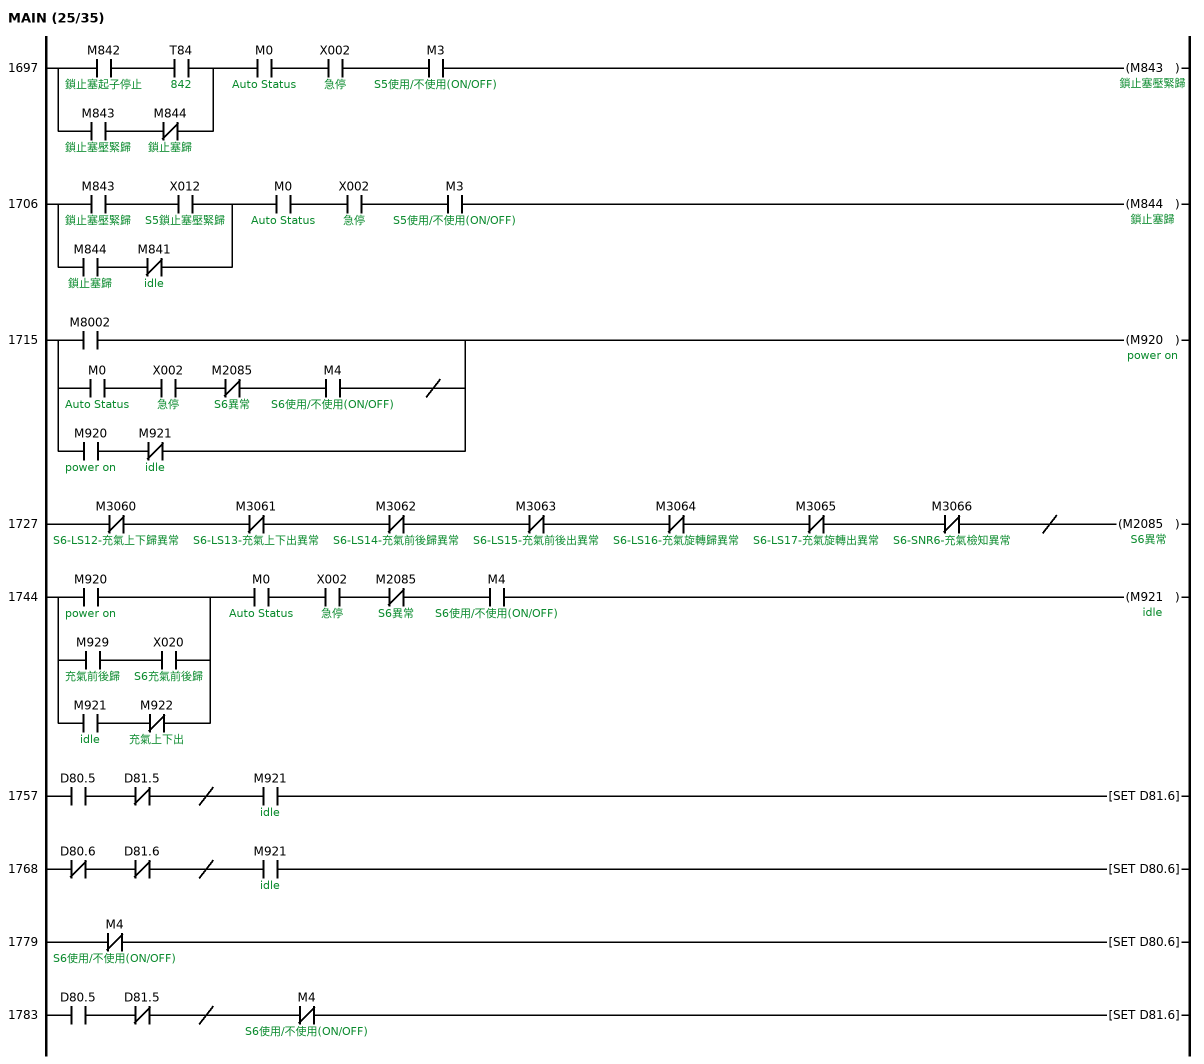
[picture p24: ladder of MAIN, rungs at steps 1697 to 1783]
1697  LD      M842  ; 鎖止塞起子停止
      AND     T84  ; 842
      LD      M843  ; 鎖止塞壓緊歸
      ANI     M844  ; 鎖止塞歸
      ORB
      AND     M0  ; Auto Status
      AND     X002  ; 急停
      AND     M3  ; S5使用/不使用(ON/OFF)
      OUT     M843  ; 鎖止塞壓緊歸
1706  LD      M843  ; 鎖止塞壓緊歸
      AND     X012  ; S5鎖止塞壓緊歸
      LD      M844  ; 鎖止塞歸
      ANI     M841  ; idle
      ORB
      AND     M0  ; Auto Status
      AND     X002  ; 急停
      AND     M3  ; S5使用/不使用(ON/OFF)
      OUT     M844  ; 鎖止塞歸
1715  LD      M8002
      LD      M0  ; Auto Status
      AND     X002  ; 急停
      ANI     M2085  ; S6異常
      AND     M4  ; S6使用/不使用(ON/OFF)
      INV
      ORB
      LD      M920  ; power on
      ANI     M921  ; idle
      ORB
      OUT     M920  ; power on
1727  LDI     M3060  ; S6-LS12-充氣上下歸異常
      ANI     M3061  ; S6-LS13-充氣上下出異常
      ANI     M3062  ; S6-LS14-充氣前後歸異常
      ANI     M3063  ; S6-LS15-充氣前後出異常
      ANI     M3064  ; S6-LS16-充氣旋轉歸異常
      ANI     M3065  ; S6-LS17-充氣旋轉出異常
      ANI     M3066  ; S6-SNR6-充氣檢知異常
      INV
      OUT     M2085  ; S6異常
1744  LD      M920  ; power on
      LD      M929  ; 充氣前後歸
      AND     X020  ; S6充氣前後歸
      ORB
      LD      M921  ; idle
      ANI     M922  ; 充氣上下出
      ORB
      AND     M0  ; Auto Status
      AND     X002  ; 急停
      ANI     M2085  ; S6異常
      AND     M4  ; S6使用/不使用(ON/OFF)
      OUT     M921  ; idle
1757  LD      D80.5
      ANI     D81.5
      INV
      AND     M921  ; idle
      SET     D81.6
1768  LDI     D80.6
      ANI     D81.6
      INV
      AND     M921  ; idle
      SET     D80.6
1779  LDI     M4  ; S6使用/不使用(ON/OFF)
      SET     D80.6
1783  LD      D80.5
      ANI     D81.5
      INV
      ANI     M4  ; S6使用/不使用(ON/OFF)
      SET     D81.6
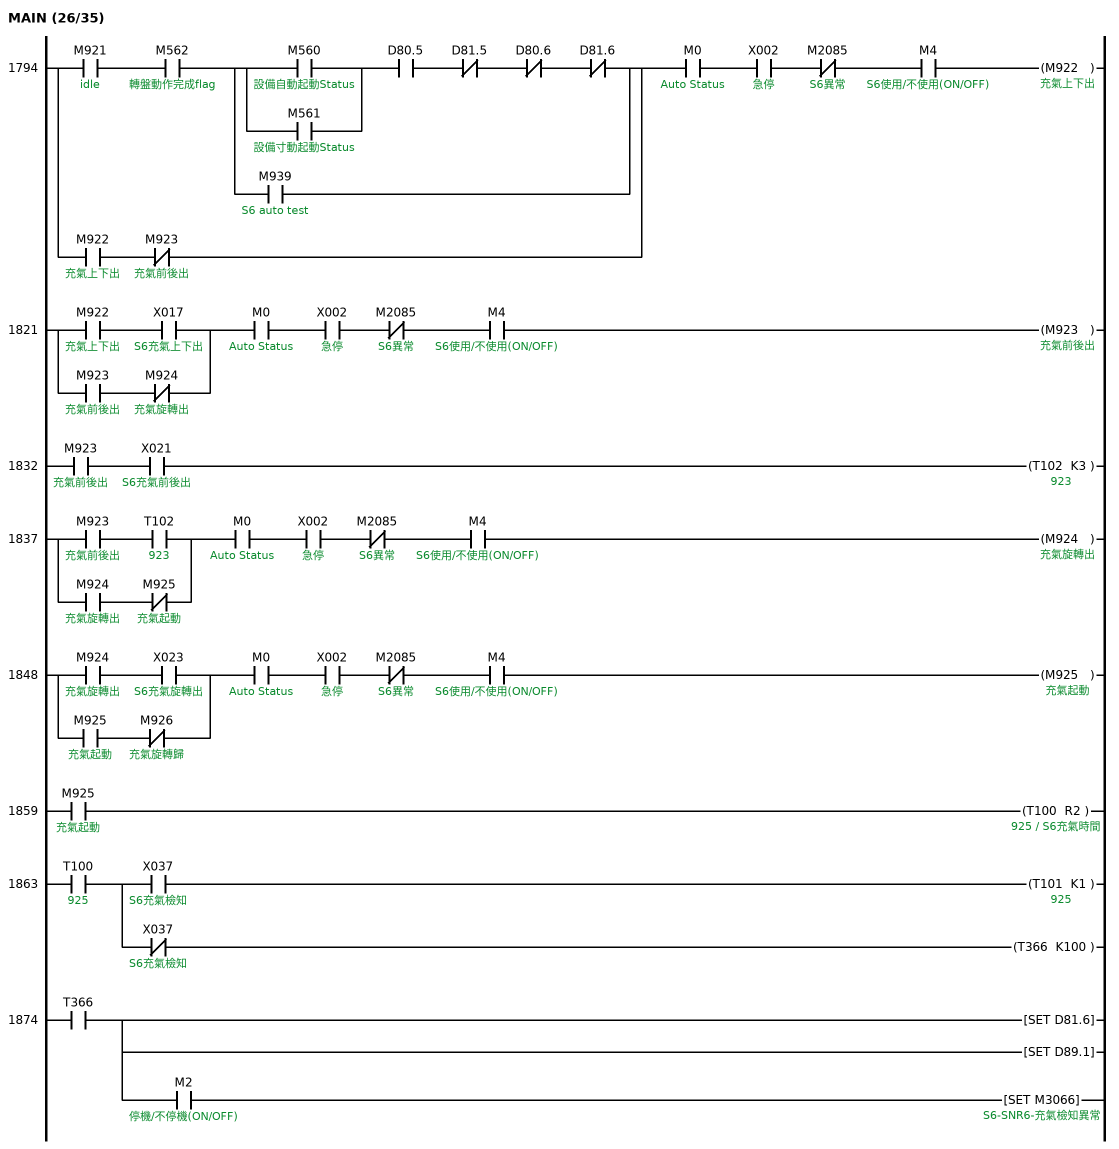
1794  LD      M921  ; idle
      AND     M562  ; 轉盤動作完成flag
      LD      M560  ; 設備自動起動Status
      OR      M561  ; 設備寸動起動Status
      AND     D80.5
      ANI     D81.5
      ANI     D80.6
      ANI     D81.6
      OR      M939  ; S6 auto test
      ANB
      LD      M922  ; 充氣上下出
      ANI     M923  ; 充氣前後出
      ORB
      AND     M0  ; Auto Status
      AND     X002  ; 急停
      ANI     M2085  ; S6異常
      AND     M4  ; S6使用/不使用(ON/OFF)
      OUT     M922  ; 充氣上下出
1821  LD      M922  ; 充氣上下出
      AND     X017  ; S6充氣上下出
      LD      M923  ; 充氣前後出
      ANI     M924  ; 充氣旋轉出
      ORB
      AND     M0  ; Auto Status
      AND     X002  ; 急停
      ANI     M2085  ; S6異常
      AND     M4  ; S6使用/不使用(ON/OFF)
      OUT     M923  ; 充氣前後出
1832  LD      M923  ; 充氣前後出
      AND     X021  ; S6充氣前後出
      OUT     T102 K3  ; 923
1837  LD      M923  ; 充氣前後出
      AND     T102  ; 923
      LD      M924  ; 充氣旋轉出
      ANI     M925  ; 充氣起動
      ORB
      AND     M0  ; Auto Status
      AND     X002  ; 急停
      ANI     M2085  ; S6異常
      AND     M4  ; S6使用/不使用(ON/OFF)
      OUT     M924  ; 充氣旋轉出
1848  LD      M924  ; 充氣旋轉出
      AND     X023  ; S6充氣旋轉出
      LD      M925  ; 充氣起動
      ANI     M926  ; 充氣旋轉歸
      ORB
      AND     M0  ; Auto Status
      AND     X002  ; 急停
      ANI     M2085  ; S6異常
      AND     M4  ; S6使用/不使用(ON/OFF)
      OUT     M925  ; 充氣起動
1859  LD      M925  ; 充氣起動
      OUT     T100 R2  ; 925 / S6充氣時間
1863  LD      T100  ; 925
      MPS
      AND     X037  ; S6充氣檢知
      OUT     T101 K1  ; 925
      MPP
      ANI     X037  ; S6充氣檢知
      OUT     T366 K100
1874  LD      T366
      SET     D81.6
      SET     D89.1
      AND     M2  ; 停機/不停機(ON/OFF)
      SET     M3066  ; S6-SNR6-充氣檢知異常
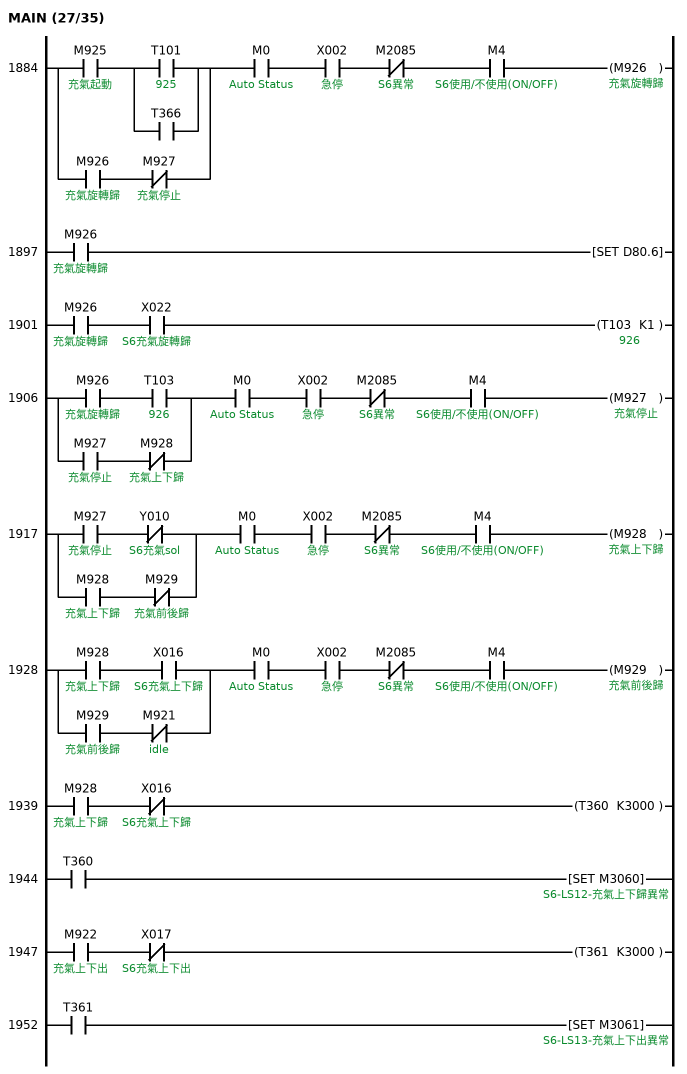
1884  LD      M925  ; 充氣起動
      LD      T101  ; 925
      OR      T366
      ANB
      LD      M926  ; 充氣旋轉歸
      ANI     M927  ; 充氣停止
      ORB
      AND     M0  ; Auto Status
      AND     X002  ; 急停
      ANI     M2085  ; S6異常
      AND     M4  ; S6使用/不使用(ON/OFF)
      OUT     M926  ; 充氣旋轉歸
1897  LD      M926  ; 充氣旋轉歸
      SET     D80.6
1901  LD      M926  ; 充氣旋轉歸
      AND     X022  ; S6充氣旋轉歸
      OUT     T103 K1  ; 926
1906  LD      M926  ; 充氣旋轉歸
      AND     T103  ; 926
      LD      M927  ; 充氣停止
      ANI     M928  ; 充氣上下歸
      ORB
      AND     M0  ; Auto Status
      AND     X002  ; 急停
      ANI     M2085  ; S6異常
      AND     M4  ; S6使用/不使用(ON/OFF)
      OUT     M927  ; 充氣停止
1917  LD      M927  ; 充氣停止
      ANI     Y010  ; S6充氣sol
      LD      M928  ; 充氣上下歸
      ANI     M929  ; 充氣前後歸
      ORB
      AND     M0  ; Auto Status
      AND     X002  ; 急停
      ANI     M2085  ; S6異常
      AND     M4  ; S6使用/不使用(ON/OFF)
      OUT     M928  ; 充氣上下歸
1928  LD      M928  ; 充氣上下歸
      AND     X016  ; S6充氣上下歸
      LD      M929  ; 充氣前後歸
      ANI     M921  ; idle
      ORB
      AND     M0  ; Auto Status
      AND     X002  ; 急停
      ANI     M2085  ; S6異常
      AND     M4  ; S6使用/不使用(ON/OFF)
      OUT     M929  ; 充氣前後歸
1939  LD      M928  ; 充氣上下歸
      ANI     X016  ; S6充氣上下歸
      OUT     T360 K3000
1944  LD      T360
      SET     M3060  ; S6-LS12-充氣上下歸異常
1947  LD      M922  ; 充氣上下出
      ANI     X017  ; S6充氣上下出
      OUT     T361 K3000
1952  LD      T361
      SET     M3061  ; S6-LS13-充氣上下出異常
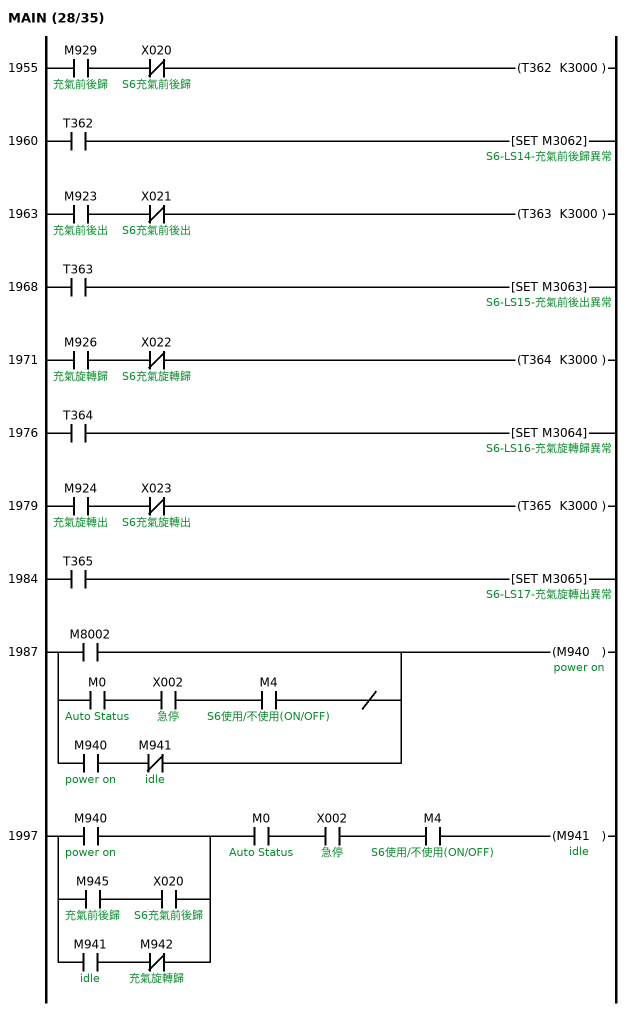
1955  LD      M929  ; 充氣前後歸
      ANI     X020  ; S6充氣前後歸
      OUT     T362 K3000
1960  LD      T362
      SET     M3062  ; S6-LS14-充氣前後歸異常
1963  LD      M923  ; 充氣前後出
      ANI     X021  ; S6充氣前後出
      OUT     T363 K3000
1968  LD      T363
      SET     M3063  ; S6-LS15-充氣前後出異常
1971  LD      M926  ; 充氣旋轉歸
      ANI     X022  ; S6充氣旋轉歸
      OUT     T364 K3000
1976  LD      T364
      SET     M3064  ; S6-LS16-充氣旋轉歸異常
1979  LD      M924  ; 充氣旋轉出
      ANI     X023  ; S6充氣旋轉出
      OUT     T365 K3000
1984  LD      T365
      SET     M3065  ; S6-LS17-充氣旋轉出異常
1987  LD      M8002
      LD      M0  ; Auto Status
      AND     X002  ; 急停
      AND     M4  ; S6使用/不使用(ON/OFF)
      INV
      ORB
      LD      M940  ; power on
      ANI     M941  ; idle
      ORB
      OUT     M940  ; power on
1997  LD      M940  ; power on
      LD      M945  ; 充氣前後歸
      AND     X020  ; S6充氣前後歸
      ORB
      LD      M941  ; idle
      ANI     M942  ; 充氣旋轉歸
      ORB
      AND     M0  ; Auto Status
      AND     X002  ; 急停
      AND     M4  ; S6使用/不使用(ON/OFF)
      OUT     M941  ; idle
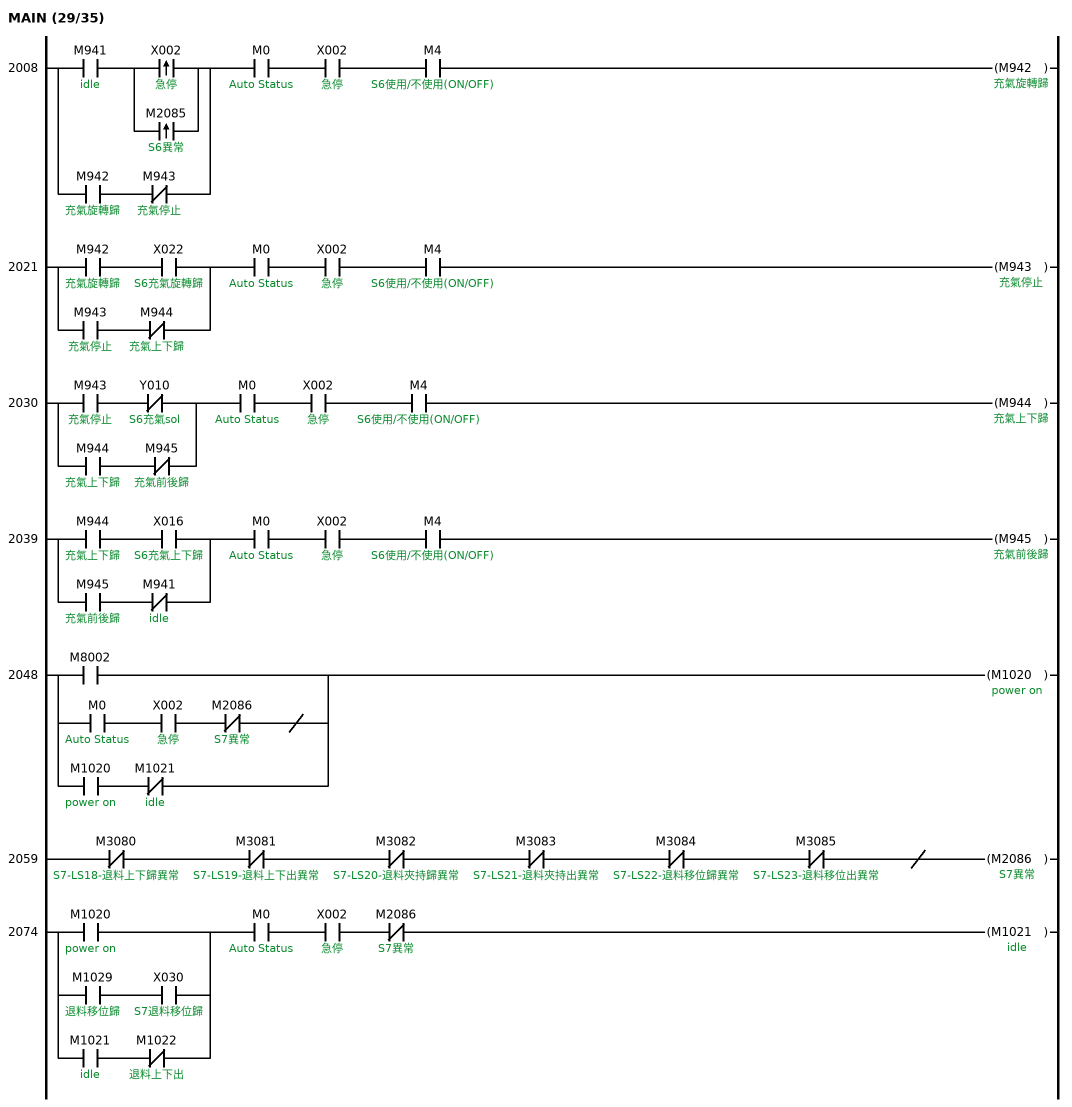
2008  LD      M941  ; idle
      LDP     X002  ; 急停
      ORP     M2085  ; S6異常
      ANB
      LD      M942  ; 充氣旋轉歸
      ANI     M943  ; 充氣停止
      ORB
      AND     M0  ; Auto Status
      AND     X002  ; 急停
      AND     M4  ; S6使用/不使用(ON/OFF)
      OUT     M942  ; 充氣旋轉歸
2021  LD      M942  ; 充氣旋轉歸
      AND     X022  ; S6充氣旋轉歸
      LD      M943  ; 充氣停止
      ANI     M944  ; 充氣上下歸
      ORB
      AND     M0  ; Auto Status
      AND     X002  ; 急停
      AND     M4  ; S6使用/不使用(ON/OFF)
      OUT     M943  ; 充氣停止
2030  LD      M943  ; 充氣停止
      ANI     Y010  ; S6充氣sol
      LD      M944  ; 充氣上下歸
      ANI     M945  ; 充氣前後歸
      ORB
      AND     M0  ; Auto Status
      AND     X002  ; 急停
      AND     M4  ; S6使用/不使用(ON/OFF)
      OUT     M944  ; 充氣上下歸
2039  LD      M944  ; 充氣上下歸
      AND     X016  ; S6充氣上下歸
      LD      M945  ; 充氣前後歸
      ANI     M941  ; idle
      ORB
      AND     M0  ; Auto Status
      AND     X002  ; 急停
      AND     M4  ; S6使用/不使用(ON/OFF)
      OUT     M945  ; 充氣前後歸
2048  LD      M8002
      LD      M0  ; Auto Status
      AND     X002  ; 急停
      ANI     M2086  ; S7異常
      INV
      ORB
      LD      M1020  ; power on
      ANI     M1021  ; idle
      ORB
      OUT     M1020  ; power on
2059  LDI     M3080  ; S7-LS18-退料上下歸異常
      ANI     M3081  ; S7-LS19-退料上下出異常
      ANI     M3082  ; S7-LS20-退料夾持歸異常
      ANI     M3083  ; S7-LS21-退料夾持出異常
      ANI     M3084  ; S7-LS22-退料移位歸異常
      ANI     M3085  ; S7-LS23-退料移位出異常
      INV
      OUT     M2086  ; S7異常
2074  LD      M1020  ; power on
      LD      M1029  ; 退料移位歸
      AND     X030  ; S7退料移位歸
      ORB
      LD      M1021  ; idle
      ANI     M1022  ; 退料上下出
      ORB
      AND     M0  ; Auto Status
      AND     X002  ; 急停
      ANI     M2086  ; S7異常
      OUT     M1021  ; idle
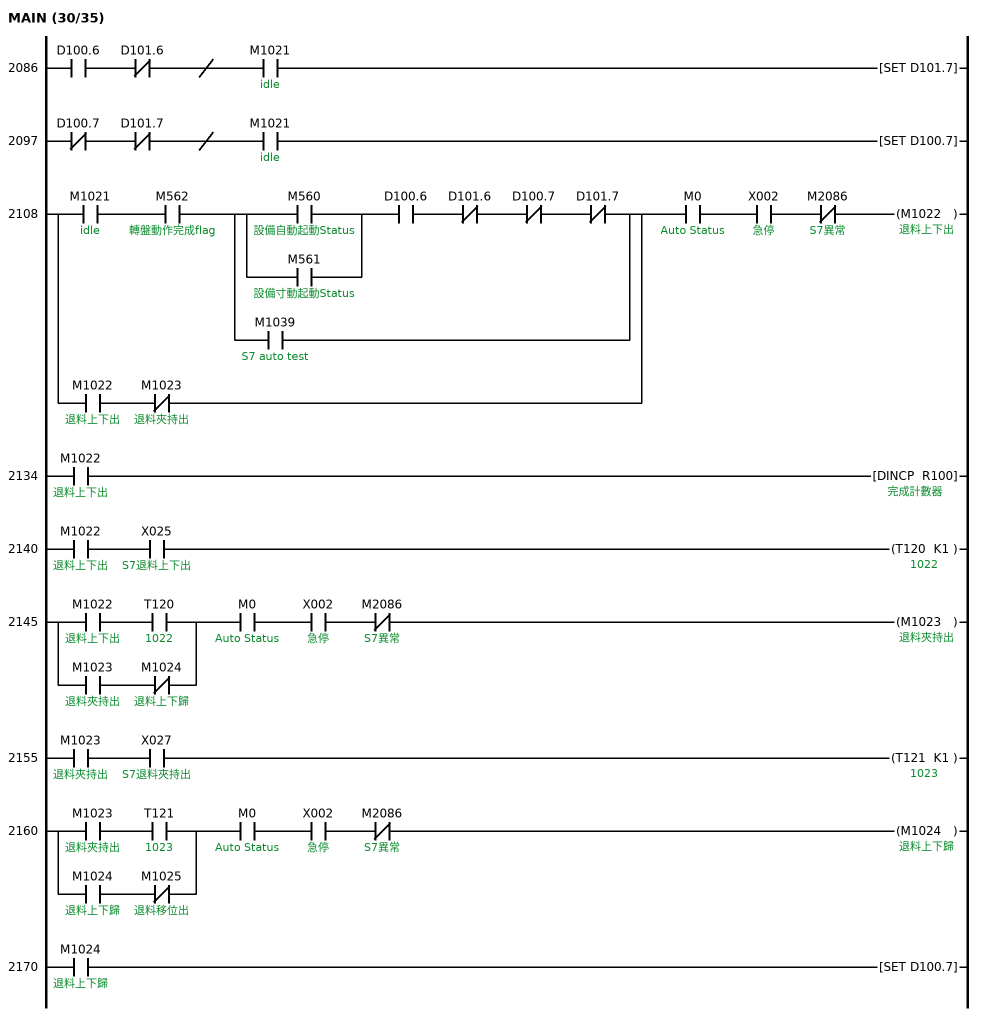
2086  LD      D100.6
      ANI     D101.6
      INV
      AND     M1021  ; idle
      SET     D101.7
2097  LDI     D100.7
      ANI     D101.7
      INV
      AND     M1021  ; idle
      SET     D100.7
2108  LD      M1021  ; idle
      AND     M562  ; 轉盤動作完成flag
      LD      M560  ; 設備自動起動Status
      OR      M561  ; 設備寸動起動Status
      AND     D100.6
      ANI     D101.6
      ANI     D100.7
      ANI     D101.7
      OR      M1039  ; S7 auto test
      ANB
      LD      M1022  ; 退料上下出
      ANI     M1023  ; 退料夾持出
      ORB
      AND     M0  ; Auto Status
      AND     X002  ; 急停
      ANI     M2086  ; S7異常
      OUT     M1022  ; 退料上下出
2134  LD      M1022  ; 退料上下出
      DINCP   R100  ; 完成計數器
2140  LD      M1022  ; 退料上下出
      AND     X025  ; S7退料上下出
      OUT     T120 K1  ; 1022
2145  LD      M1022  ; 退料上下出
      AND     T120  ; 1022
      LD      M1023  ; 退料夾持出
      ANI     M1024  ; 退料上下歸
      ORB
      AND     M0  ; Auto Status
      AND     X002  ; 急停
      ANI     M2086  ; S7異常
      OUT     M1023  ; 退料夾持出
2155  LD      M1023  ; 退料夾持出
      AND     X027  ; S7退料夾持出
      OUT     T121 K1  ; 1023
2160  LD      M1023  ; 退料夾持出
      AND     T121  ; 1023
      LD      M1024  ; 退料上下歸
      ANI     M1025  ; 退料移位出
      ORB
      AND     M0  ; Auto Status
      AND     X002  ; 急停
      ANI     M2086  ; S7異常
      OUT     M1024  ; 退料上下歸
2170  LD      M1024  ; 退料上下歸
      SET     D100.7
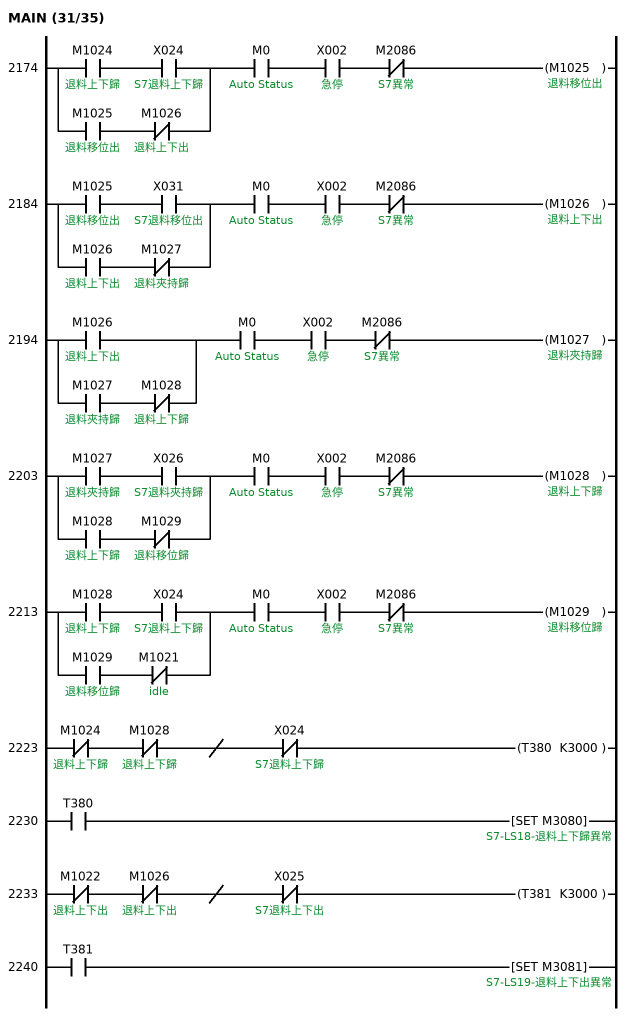
2174  LD      M1024  ; 退料上下歸
      AND     X024  ; S7退料上下歸
      LD      M1025  ; 退料移位出
      ANI     M1026  ; 退料上下出
      ORB
      AND     M0  ; Auto Status
      AND     X002  ; 急停
      ANI     M2086  ; S7異常
      OUT     M1025  ; 退料移位出
2184  LD      M1025  ; 退料移位出
      AND     X031  ; S7退料移位出
      LD      M1026  ; 退料上下出
      ANI     M1027  ; 退料夾持歸
      ORB
      AND     M0  ; Auto Status
      AND     X002  ; 急停
      ANI     M2086  ; S7異常
      OUT     M1026  ; 退料上下出
2194  LD      M1026  ; 退料上下出
      LD      M1027  ; 退料夾持歸
      ANI     M1028  ; 退料上下歸
      ORB
      AND     M0  ; Auto Status
      AND     X002  ; 急停
      ANI     M2086  ; S7異常
      OUT     M1027  ; 退料夾持歸
2203  LD      M1027  ; 退料夾持歸
      AND     X026  ; S7退料夾持歸
      LD      M1028  ; 退料上下歸
      ANI     M1029  ; 退料移位歸
      ORB
      AND     M0  ; Auto Status
      AND     X002  ; 急停
      ANI     M2086  ; S7異常
      OUT     M1028  ; 退料上下歸
2213  LD      M1028  ; 退料上下歸
      AND     X024  ; S7退料上下歸
      LD      M1029  ; 退料移位歸
      ANI     M1021  ; idle
      ORB
      AND     M0  ; Auto Status
      AND     X002  ; 急停
      ANI     M2086  ; S7異常
      OUT     M1029  ; 退料移位歸
2223  LDI     M1024  ; 退料上下歸
      ANI     M1028  ; 退料上下歸
      INV
      ANI     X024  ; S7退料上下歸
      OUT     T380 K3000
2230  LD      T380
      SET     M3080  ; S7-LS18-退料上下歸異常
2233  LDI     M1022  ; 退料上下出
      ANI     M1026  ; 退料上下出
      INV
      ANI     X025  ; S7退料上下出
      OUT     T381 K3000
2240  LD      T381
      SET     M3081  ; S7-LS19-退料上下出異常
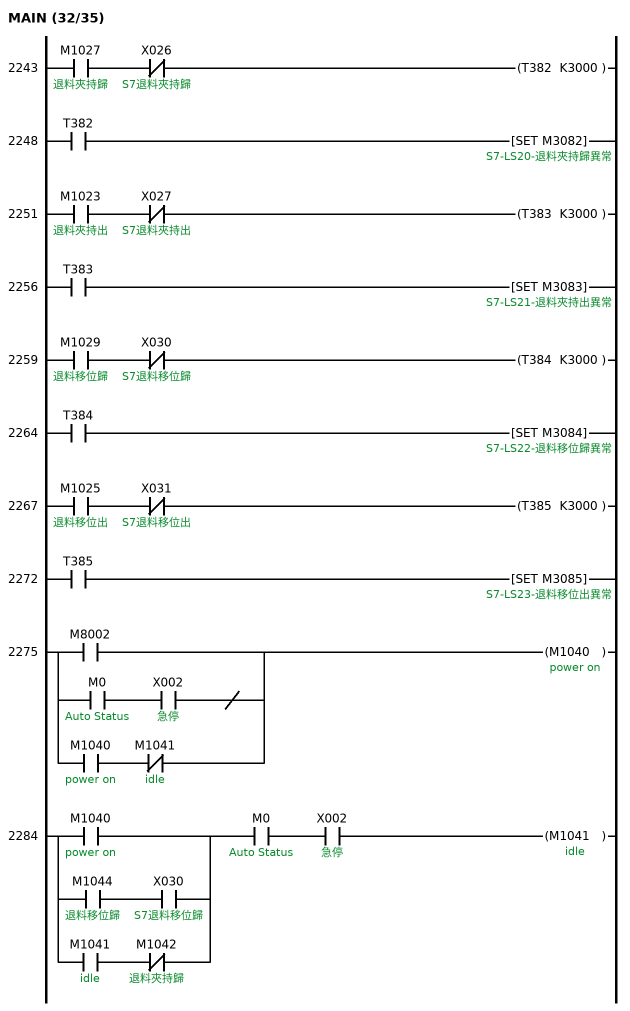
2243  LD      M1027  ; 退料夾持歸
      ANI     X026  ; S7退料夾持歸
      OUT     T382 K3000
2248  LD      T382
      SET     M3082  ; S7-LS20-退料夾持歸異常
2251  LD      M1023  ; 退料夾持出
      ANI     X027  ; S7退料夾持出
      OUT     T383 K3000
2256  LD      T383
      SET     M3083  ; S7-LS21-退料夾持出異常
2259  LD      M1029  ; 退料移位歸
      ANI     X030  ; S7退料移位歸
      OUT     T384 K3000
2264  LD      T384
      SET     M3084  ; S7-LS22-退料移位歸異常
2267  LD      M1025  ; 退料移位出
      ANI     X031  ; S7退料移位出
      OUT     T385 K3000
2272  LD      T385
      SET     M3085  ; S7-LS23-退料移位出異常
2275  LD      M8002
      LD      M0  ; Auto Status
      AND     X002  ; 急停
      INV
      ORB
      LD      M1040  ; power on
      ANI     M1041  ; idle
      ORB
      OUT     M1040  ; power on
2284  LD      M1040  ; power on
      LD      M1044  ; 退料移位歸
      AND     X030  ; S7退料移位歸
      ORB
      LD      M1041  ; idle
      ANI     M1042  ; 退料夾持歸
      ORB
      AND     M0  ; Auto Status
      AND     X002  ; 急停
      OUT     M1041  ; idle
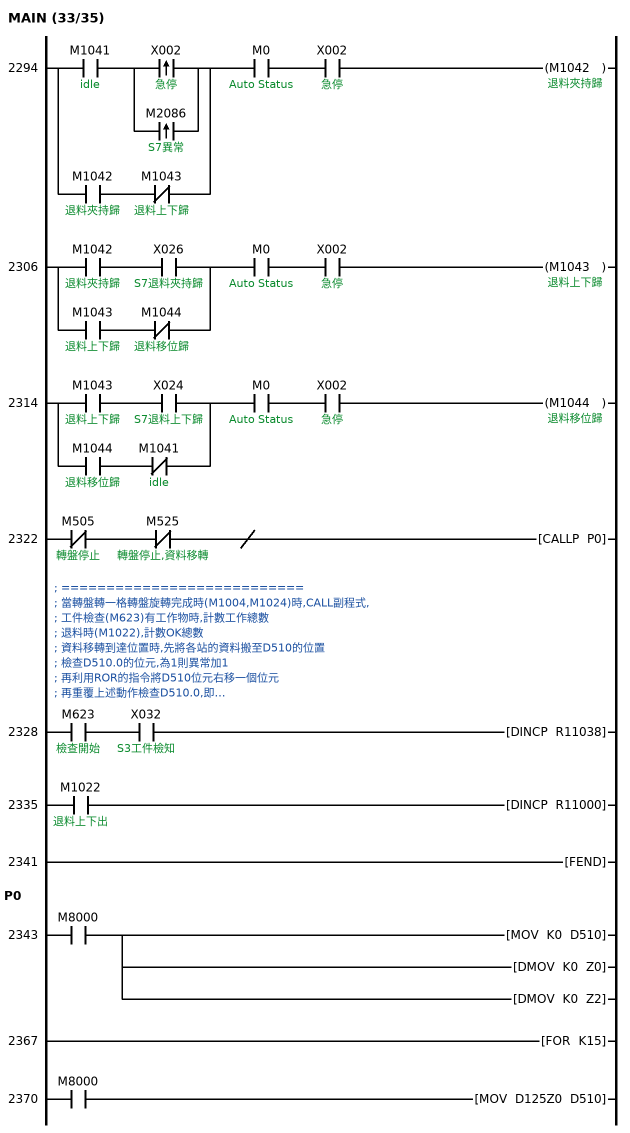
2294  LD      M1041  ; idle
      LDP     X002  ; 急停
      ORP     M2086  ; S7異常
      ANB
      LD      M1042  ; 退料夾持歸
      ANI     M1043  ; 退料上下歸
      ORB
      AND     M0  ; Auto Status
      AND     X002  ; 急停
      OUT     M1042  ; 退料夾持歸
2306  LD      M1042  ; 退料夾持歸
      AND     X026  ; S7退料夾持歸
      LD      M1043  ; 退料上下歸
      ANI     M1044  ; 退料移位歸
      ORB
      AND     M0  ; Auto Status
      AND     X002  ; 急停
      OUT     M1043  ; 退料上下歸
2314  LD      M1043  ; 退料上下歸
      AND     X024  ; S7退料上下歸
      LD      M1044  ; 退料移位歸
      ANI     M1041  ; idle
      ORB
      AND     M0  ; Auto Status
      AND     X002  ; 急停
      OUT     M1044  ; 退料移位歸
2322  LDI     M505  ; 轉盤停止
      ANI     M525  ; 轉盤停止,資料移轉
      INV
      CALLP   P0
; ===========================
; 當轉盤轉一格轉盤旋轉完成時(M1004,M1024)時,CALL副程式,
; 工件檢查(M623)有工作物時,計數工作總數
; 退料時(M1022),計數OK總數
; 資料移轉到達位置時,先將各站的資料搬至D510的位置
; 檢查D510.0的位元,為1則異常加1
; 再利用ROR的指令將D510位元右移一個位元
; 再重覆上述動作檢查D510.0,即可
; 故要利用此程式只要改變IDLE(M1001,M1021),各站異常區(D145)
; D510,D520,和資料表R10000~R10299在主程式不要佔用到不然也要變更
; P0的程式放在主程式最尾端
; ===========================
2328  LD      M623  ; 檢查開始
      AND     X032  ; S3工件檢知
      DINCP   R11038
2335  LD      M1022  ; 退料上下出
      DINCP   R11000
2341  FEND
      P0
2343  LD      M8000
      MOV     K0 D510
      DMOV    K0 Z0
      DMOV    K0 Z2
2367  FOR     K15
2370  LD      M8000
      MOV     D125Z0 D510
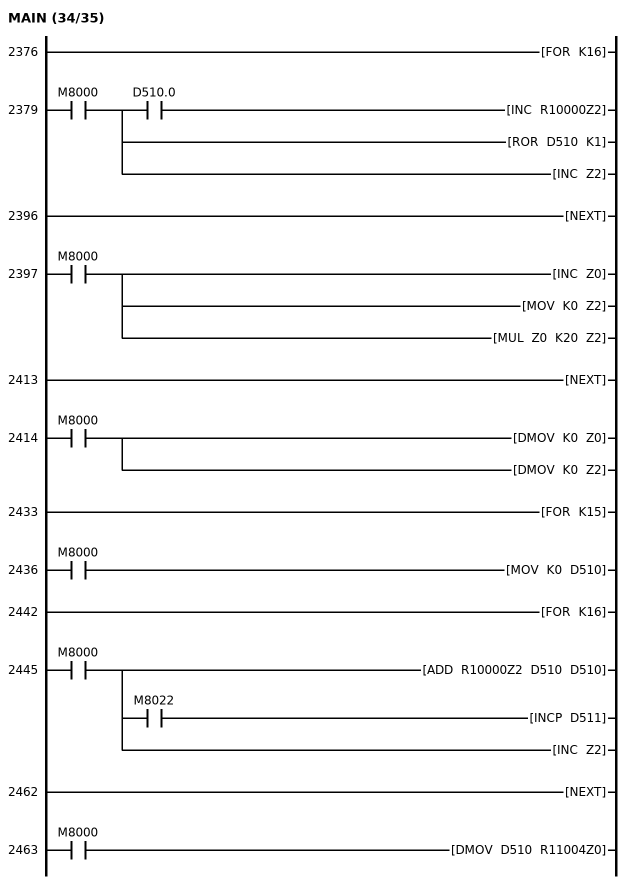
2376  FOR     K16
2379  LD      M8000
      MPS
      AND     D510.0
      INC     R10000Z2
      MPP
      ROR     D510 K1
      INC     Z2
2396  NEXT
2397  LD      M8000
      INC     Z0
      MOV     K0 Z2
      MUL     Z0 K20 Z2
2413  NEXT
2414  LD      M8000
      DMOV    K0 Z0
      DMOV    K0 Z2
2433  FOR     K15
2436  LD      M8000
      MOV     K0 D510
2442  FOR     K16
2445  LD      M8000
      ADD     R10000Z2 D510 D510
      MPS
      AND     M8022
      INCP    D511
      MPP
      INC     Z2
2462  NEXT
2463  LD      M8000
      DMOV    D510 R11004Z0
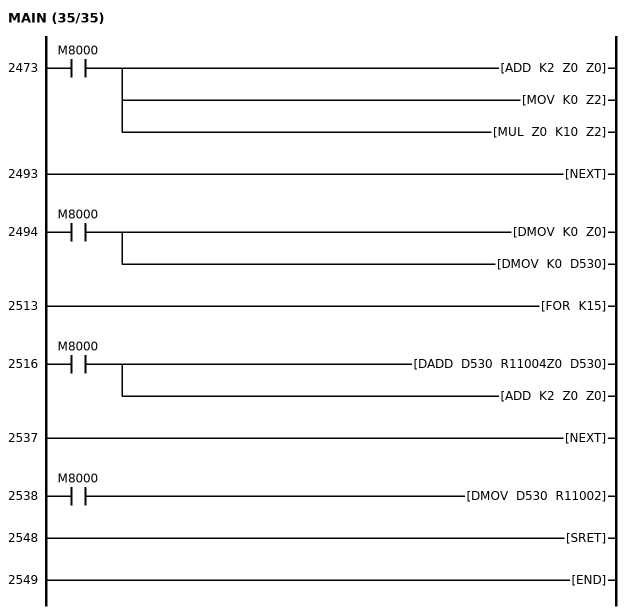
2473  LD      M8000
      ADD     K2 Z0 Z0
      MOV     K0 Z2
      MUL     Z0 K10 Z2
2493  NEXT
2494  LD      M8000
      DMOV    K0 Z0
      DMOV    K0 D530
2513  FOR     K15
2516  LD      M8000
      DADD    D530 R11004Z0 D530
      ADD     K2 Z0 Z0
2537  NEXT
2538  LD      M8000
      DMOV    D530 R11002
2548  SRET
2549  END
END_PROGRAM

// device comments not shown above
D145  ; #1第2站QC
M570  ; 統計清除
M630  ; 噴油選擇
M3025  ; S4-SNR3-旋塞浮鎖檢知異常
Y025  ; 轉盤馬達電源
D1  ; #2NG狀態
D2  ; #2動作狀態
D5  ; #2第2站QC
D6  ; #2第3站QC
D7  ; #2第4站QC
D8  ; #2第5站QC
D9  ; #2第6站QC
D10  ; #2第7站QC
D11  ; #2第8站QC
D20  ; #3完成狀態
D21  ; #3NG狀態
D22  ; #3動作狀態
D25  ; #3第2站QC
D26  ; #3第3站QC
D27  ; #3第4站QC
D28  ; #3第5站QC
D29  ; #3第6站QC
D30  ; #3第7站QC
D31  ; #3第8站QC
D40  ; #4完成狀態
D41  ; #4NG狀態
D42  ; #4動作狀態
D45  ; #4第2站QC
D46  ; #4第3站QC
D47  ; #4第4站QC
D48  ; #4第5站QC
D49  ; #4第6站QC
D50  ; #4第7站QC
D51  ; #4第8站QC
D60  ; #5完成狀態
D61  ; #5NG狀態
D62  ; #5動作狀態
D65  ; #5第2站QC
D66  ; #5第3站QC
D67  ; #5第4站QC
D68  ; #5第5站QC
D69  ; #5第6站QC
D70  ; #5第7站QC
D71  ; #5第8站QC
D80  ; #6完成狀態
D81  ; #6NG狀態
D82  ; #6動作狀態
D85  ; #6第2站QC
D86  ; #6第3站QC
D87  ; #6第4站QC
D88  ; #6第5站QC
D89  ; #6第6站QC
D90  ; #6第7站QC
D91  ; #6第8站QC
D100  ; #7完成狀態
D101  ; #7NG狀態
D102  ; #7動作狀態
D105  ; #7第2站QC
D106  ; #7第3站QC
D107  ; #7第4站QC
D108  ; #7第5站QC
D109  ; #7第6站QC
D110  ; #7第7站QC
D111  ; #7第8站QC
D121  ; #8NG狀態
D122  ; #8動作狀態
D125  ; #8第2站QC
D127  ; #8第4站QC
D129  ; #8第6站QC
D131  ; #8第8站QC
D140  ; #1完成狀態
D141  ; #1NG狀態
D142  ; #1動作狀態
D146  ; #1第3站QC
D147  ; #1第4站QC
D148  ; #1第5站QC
D149  ; #1第6站QC
D150  ; #1第7站QC
D151  ; #1第8站QC
T13  ; S7退料移位歸sol
T14  ; S7退料移位出sol
T15  ; 轉盤馬達運轉relay
